{attribute 'qualified_only'}
VAR_GLOBAL
	K1	 AT %Q*:BOOL;     // 	Aktor Füllung
	K2	 AT %Q*:BOOL;     // 	Aktor Vereinzelung
	P1	 AT %Q*:BOOL;     // 	 Anlage Ein
	P2	 AT %Q*:BOOL;     // 	Meldeleuchte STörung
	Q1	 AT %Q*:BOOL;     // 	Antrieb Förderband
END_VAR

(* stored: Version 1.1.0.1, ProductVersion 3.1.4024.5
   GVL DA: Id {efa3d63a-96e1-4204-b1e7-9f3703bd4f03} *)
